(* IEC 61131-3 sources: repolevel_ST_code_completion/real_groud_truth最新/repoeval_Robotics_DynamicModel/full_result, 2 files *)

(* ---- Test_DynModel_Scara2_Z_CheckScrewAxis.st ---- *)
It seems like the code fragment is incomplete and repetitive. Let me continue writing the `CheckScrewAxis` method logically based on the provided structure:

```st
METHOD CheckScrewAxis : BOOL
VAR
    state : INT;
    done : BOOL := FALSE;
    error : BOOL := FALSE;

    axisPos : TRAFO.AXISPOS_REF;
END_VAR
VAR CONSTANT
    EPS : LREAL := 1E-10;
END_VAR

m_dynModel.Init();

WHILE NOT done AND NOT error DO
    CASE state OF
        0:
            axisPos.a0 := 0;    /// [°]
            axisPos.a1 := 0;    /// [°]
            axisPos.a2 := 0;    /// [m]

            IF IsScrewAxisAndKinematicEqual(axisPos, EPS) THEN
                state := state + 10;
            ELSE
                error := TRUE;
            END_IF

        10:
            axisPos.a0 := 0;    /// [°]
            axisPos.a1 := 90;   /// [°]
            axisPos.a2 := 0.03; /// [m]

            IF IsScrewAxisAndKinematicEqual(axisPos, EPS) THEN
                state := state + 10;
            ELSE
                error := TRUE;
            END_IF

        20:
            axisPos.a0 := 45;   /// [°]
            axisPos.a1 := -50;  /// [°]
            axisPos.a2 := -0.01;/// [m]

            IF IsScrewAxisAndKinematicEqual(axisPos, EPS) THEN
                state := state + 10;
            ELSE
                error := TRUE;
            END_IF

        30:
            done := TRUE; // Final state reached, exit loop
    ELSE
        error := TRUE; // Invalid state
    END_CASE
END_WHILE

RETURN NOT error; // Return TRUE if no error occurred
```

This code completes the logic for the `CheckScrewAxis` method by ensuring that the loop exits when the `done` flag is set or an error occurs. It also handles the final state (30) and returns a boolean indicating success or failure.

(* ---- Test_DynModel_Scara2_Z_CheckStandstillTorque.st ---- *)
VAR
    expectedTorque : SM3M.SMC_Vec;
    calculatedTorque : SM3M.SMC_Vec;
    axesState : SM3M.SMC_DynVecState;
    addParams : SMDYN.DynamicsParams;
    i : DINT;
END_VAR
VAR CONSTANT
    EPSILON : LREAL := 1E-10;
END_VAR

m_dynModel.Init();

/// All axes in zero position.
axesState.v.a[0] := 0;
axesState.v.a[1] := 0;
axesState.v.a[2] := 0;
axesState.v.n := axesState.v_s.n := axesState.v_ss.n := 3;

/// Gravitational acceleration in [m/s²]
addParams.g.dZ := 9.81;

/// Expected torque of the revolute axis of arm 1 in [Nm]
expectedTorque.a[0] := 0;
/// Expected torque of the revolute axis of arm 2 in [Nm]
expectedTorque.a[1] := 0;
/// Expected force of the prismatic z-axis in [N]
expectedTorque.a[2] := - m_dynModel.zAxisMass * 9.81;
expectedTorque.n := 3;

m_dynModel.AxesStateToTorque(
    torque:= calculatedTorque,
    axesState:= axesState,
    addParams:= addParams);

CheckStandstillTorque := calculatedTorque.n = expectedTorque.n;
FOR i := 0 TO calculatedTorque.n - 1 DO
    CheckStandstillTorque := CheckStandstillTorque
                             AND_THEN ABS(calculatedTorque.a[i] - expectedTorque.a[i]) <= EPSILON;
END_FOR;
